# EPICS autosave request: ADCore/ADApp/Db/NDColorConvert_settings.req
$(P)$(R)ColorModeOut
